(* PLC project spsna002.project, CODESYS CODESYS V3.5 SP21 Patch 2 *)
(* stored: creationDateTime 2025-10-28T20:53:01.1932882, modificationDateTime 2025-10-28T20:42:45.2900829 *)

TYPE SControlWord_t : STRUCT
  Enable : BOOL;
  Start : BOOL;
  Stop : BOOL;
  Direction : BOOL;
END_STRUCT;
END_TYPE

TYPE SStatusWord_t : STRUCT
  Enable : BOOL;
  Stop : BOOL;
  Direction : BOOL;
  N0 : BOOL;
END_STRUCT;
END_TYPE

PROGRAM PLC_PRG
  VAR
    Inverter : FB_Inverter;
  END_VAR

                    

Inverter(
	enable := GlobalVariable.Freigabe, 
	setPoint	:= GlobalVariable.Sollwert,
	controlWord := GlobalVariable.SteuerWort,
	actValue => GlobalVariable.Istwert,
	statusWord => GlobalVariable.StatusWort
);


                  
END_PROGRAM

FUNCTION_BLOCK FB_Inverter
  VAR_INPUT
    enable : BOOL;
    setPoint : REAL;
    controlWord : SControlWord_t;
    rampUp : REAL := 10.0;
    rampDown : REAL := 5.0;
  END_VAR
  VAR_OUTPUT
    actValue : REAL;
    statusWord : SStatusWord_t;
    actPosition : REAL;
  END_VAR
  VAR
    rampSpeedUp : REAL;
    rampSpeedDown : REAL;
  END_VAR

                    


  
IF enable THEN


	
	IF rampUp > 0.0 THEN
		rampSpeedUp := (GlobaleConstants.MAX_SET_POINT - GlobaleConstants.MIN_SET_POINT) / rampUp;
	ELSE
		rampSpeedUp := 999999.0;
	END_IF


	IF rampDown > 0.0 THEN
		rampSpeedDown := (GlobaleConstants.MAX_SET_POINT - GlobaleConstants.MIN_SET_POINT) / rampDown;
	ELSE
		rampSpeedDown := 999999.0;
	END_IF


	setPoint := LIMIT(GlobaleConstants.MIN_SET_POINT, setPoint, GlobaleConstants.MAX_SET_POINT);

	IF controlWord.Enable THEN
	
		IF controlWord.Stop THEN
			actValue := 0.0;
		ELSIF controlWord.Start THEN
			IF setPoint > actValue THEN
				actValue := actValue + rampSpeedUp * GlobaleConstants.CYCLETIME;
				IF actValue > setPoint THEN
					actValue := setPoint;
				END_IF
			
			ELSIF setPoint < actValue THEN
				actValue := actValue - rampSpeedDown * GlobaleConstants.CYCLETIME;
				IF actValue < setPoint THEN
					actValue := setPoint;
				END_IF
			END_IF
			//actValue := setPoint;
		ELSE
			actValue := 0.0;
		END_IF
	
		IF controlWord.Direction THEN
			actValue := setPoint * -1.0;
		END_IF
		
	
	ELSE
		actValue := 0.0;
	END_IF

	statusWord.Enable := controlWord.Enable;
	statusWord.Stop := controlWord.Stop;
	statusWord.N0 := (actValue <= 0.001 AND actValue >= -0.001);

ELSE

	actValue := 0.0;
	statusWord.Enable := FALSE;
	statusWord.Stop := TRUE;
	statusWord.N0 := TRUE;

END_IF 

statusWord.Direction := controlWord.Direction;

                  
END_FUNCTION_BLOCK

CONFIGURATION Device
  RESOURCE Application ON PLC
    {attribute 'qualified_only'}
    VAR_GLOBAL  (* GlobalVariable *)
      SteuerWort : SControlWord_t;
      StatusWort : SStatusWord_t;
      Sollwert : REAL;
      Istwert : REAL;
      Freigabe : BOOL;
    END_VAR
    {attribute 'qualified_only'}
    VAR_GLOBAL CONSTANT  (* GlobaleConstants *)
      MAX_SET_POINT : REAL := 1600.0;
      MIN_SET_POINT : REAL := -1600.0;
      CYCLETIME : REAL := 0.02;
    END_VAR
    TASK MainTask(INTERVAL := T#20ms, PRIORITY := 1);
    TASK VISU_TASK(INTERVAL := T#100ms, PRIORITY := 31);
    PROGRAM PLC_PRG WITH MainTask : PLC_PRG;
    PROGRAM VisuElems.Visu_Prg WITH VISU_TASK : VisuElems.Visu_Prg;
  END_RESOURCE
END_CONFIGURATION
